										RIBALTINO_DOPO_SQUADRO:
											IF vo = 0 THEN 							
												Mission^.ZPlace			:= 	//WorkArea^[Mission^.PPlace].Z + 
																			Forming^[WorkAreaState^[cwa].F].PackXP[WorkAreaState^[cwa].P].Z + 
																			Forming^[WorkAreaState^[cwa].F].PLZ + 
																			Forming^[WorkAreaState^[cwa].F].PIZ +
																			WorkArea^[Mission^.PPlace].HPL + 
																			HalfPackDim + 
																			ZOffsetPlace + 
																			PickPlaceParameters^.OffsetZPlacePaccoVerticale +
																			DifferenceRealNominalDimensionZ/2;
											(* Quota di deposito Z con pacco orrizontale *)	
											ELSE
												Mission^.ZPlace			:= 	//WorkArea^[Mission^.PPlace].Z + 
																			Forming^[WorkAreaState^[cwa].F].PackXP[WorkAreaState^[cwa].P].Z + 
																			Forming^[WorkAreaState^[cwa].F].PLZ + 
																			WorkArea^[Mission^.PPlace].HPL + 
																			HalfPackDim + 
																			ZOffsetPlace + 
																			PickPlaceParameters^.OffsetZPlacePaccoOrrizzontale;
																			//DifferenceRealNominalDimensionZ/2;
											END_IF
									
										RIBALTINO_DIRETTO:
											IF vo = 0 THEN 							
												Mission^.ZPlace			:= 	//WorkArea^[Mission^.PPlace].Z + 
																			Forming^[WorkAreaState^[cwa].F].PackXP[WorkAreaState^[cwa].P].Z + 
																			Forming^[WorkAreaState^[cwa].F].PLZ + 
																			Forming^[WorkAreaState^[cwa].F].PIZ +
																			WorkArea^[Mission^.PPlace].HPL + 
																			Mission^.XDiM/2 + 
																			ZOffsetPlace + 
																			PickPlaceParameters^.OffsetZPlacePaccoVerticale +
																			DifferenceRealNominalDimensionZ/2;
											(* Quota di deposito Z con pacco orrizontale *)	
											ELSE
												Mission^.ZPlace			:= 	//WorkArea^[Mission^.PPlace].Z + 
																			Forming^[WorkAreaState^[cwa].F].PackXP[WorkAreaState^[cwa].P].Z + 
																			Forming^[WorkAreaState^[cwa].F].PLZ + 
																			WorkArea^[Mission^.PPlace].HPL + 
																			Mission^.ZDim/2 + 
																			ZOffsetPlace + 
																			PickPlaceParameters^.OffsetZPlacePaccoOrrizzontale +
																			DifferenceRealNominalDimensionZ/2;
											END_IF
									END_CASE
									//Mission^.ZPlace			:= WorkArea^[Mission^.PPlace].Z + Forming^[WorkAreaState^[cwa].F].PackXN[WorkAreaState^[cwa].P].Z*2 + WorkArea^[Mission^.PPlace].H;
									Mission^.JPlace			:= 	WorkArea^[Mission^.PPlace].J + 
																WorkAreaOffset^[Mission^.PPlace].J + 
																Forming^[WorkAreaState^[cwa].F].PackXP[WorkAreaState^[cwa].P].J-
																(90*(1-JP)); //x deposito con prelievo TRASVERSALE
									CASE VERSO_PALLETTIZZATORE OF 
										
										PALLETTIZZATORE_DX:
											Mission^.JPlace	:= 	WorkArea^[Mission^.PPlace].J + 
																WorkAreaOffset^[Mission^.PPlace].J + 
																Forming^[WorkAreaState^[cwa].F].PackXP[WorkAreaState^[cwa].P].J-
																(90*(1-JP));
														
										PALLETTIZZATORE_SX:
											Mission^.JPlace	:= 	WorkArea^[Mission^.PPlace].J + 
																WorkAreaOffset^[Mission^.PPlace].J + 
																Forming^[WorkAreaState^[cwa].F].PackXP[WorkAreaState^[cwa].P].J-
																(90*(1-JP));

									END_CASE							
																
																
									IF NOT SimulazioneSenzaPallet THEN //Se non sono in simulazione utilizzo la presa con coppia							
										Mission^.KPlace			:= 	kpick; (*+ 
																PickPlaceParameters^.OffsetKPlacePack;*) // Aggiungere Eventuale Offset x Apertura e Rilascio
									ELSE
										Mission^.KPlace			:= 	kpick + PickPlaceParameters^.OffsetKPickPack;
									END_IF
									Mission^.KPlaceMode 	:= 	KTORQUEMODE;
									(* Quota di Approccio con pacco verticale *)							
									IF (vo = 0 AND DisabilitaApproccioPacciOrrizzontali) OR NOT DisabilitaApproccioPacciOrrizzontali THEN 
										IF  Forming^[WorkAreaState^[cwa].F].PackXP[WorkAreaState^[cwa].P].Trajectory = 0 THEN
											Mission^.XPlaceApproach	:= Mission^.XPlace;
											Mission^.YPlaceApproach	:= Mission^.YPlace;
											Mission^.ZPlaceApproach	:= Mission^.ZPlace;
											Mission^.JPlaceApproach	:= Mission^.JPlace;
										ELSIF  Forming^[WorkAreaState^[cwa].F].PackXP[WorkAreaState^[cwa].P].Trajectory = 1 THEN	
											Mission^.XPlaceApproach	:= 	Mission^.XPlace - 
																		Forming^[WorkAreaState^[cwa].F].AX;
											Mission^.YPlaceApproach	:= 	Mission^.YPlace - 
																		Forming^[WorkAreaState^[cwa].F].AY;
											Mission^.ZPlaceApproach	:= 	Mission^.ZPlace + 
																		Forming^[WorkAreaState^[cwa].F].AZ;
											Mission^.JPlaceApproach	:= 	Mission^.JPlace;
										ELSIF  Forming^[WorkAreaState^[cwa].F].PackXP[WorkAreaState^[cwa].P].Trajectory = 111 THEN	
											Mission^.XPlaceApproach	:= 	Mission^.XPlace - 
																		Forming^[WorkAreaState^[cwa].F].AX;
											Mission^.YPlaceApproach	:= 	Mission^.YPlace - 
																		Forming^[WorkAreaState^[cwa].F].AY;
											Mission^.ZPlaceApproach	:= 	Mission^.ZPlace + 
																		Forming^[WorkAreaState^[cwa].F].AZ;
											Mission^.JPlaceApproach	:= 	Mission^.JPlace;
										ELSIF  Forming^[WorkAreaState^[cwa].F].PackXP[WorkAreaState^[cwa].P].Trajectory = 2 THEN	
											Mission^.XPlaceApproach	:= 	Mission^.XPlace + 
																		Forming^[WorkAreaState^[cwa].F].AX;
											Mission^.YPlaceApproach	:= 	Mission^.YPlace - 
																		Forming^[WorkAreaState^[cwa].F].AY;
											Mission^.ZPlaceApproach	:= 	Mission^.ZPlace + 
																		Forming^[WorkAreaState^[cwa].F].AZ;
											Mission^.JPlaceApproach	:= 	Mission^.JPlace;
										ELSIF  Forming^[WorkAreaState^[cwa].F].PackXP[WorkAreaState^[cwa].P].Trajectory = 101 THEN	
											Mission^.XPlaceApproach	:= 	Mission^.XPlace + 
																		Forming^[WorkAreaState^[cwa].F].AX;
											Mission^.YPlaceApproach	:= 	Mission^.YPlace - 
																		Forming^[WorkAreaState^[cwa].F].AY;
											Mission^.ZPlaceApproach	:= 	Mission^.ZPlace + 
																		Forming^[WorkAreaState^[cwa].F].AZ;
											Mission^.JPlaceApproach	:= 	Mission^.JPlace;
										ELSIF  Forming^[WorkAreaState^[cwa].F].PackXP[WorkAreaState^[cwa].P].Trajectory = 101 THEN	
											Mission^.XPlaceApproach	:= 	Mission^.XPlace + 
																		Forming^[WorkAreaState^[cwa].F].AX;
											Mission^.YPlaceApproach	:= 	Mission^.YPlace - 
																		Forming^[WorkAreaState^[cwa].F].AY;
											Mission^.ZPlaceApproach	:= 	Mission^.ZPlace + 
																		Forming^[WorkAreaState^[cwa].F].AZ;
											Mission^.JPlaceApproach	:= 	Mission^.JPlace;
										ELSIF  Forming^[WorkAreaState^[cwa].F].PackXP[WorkAreaState^[cwa].P].Trajectory = 201 THEN	
											Mission^.XPlaceApproach	:= 	Mission^.XPlace - 
																		Forming^[WorkAreaState^[cwa].F].AX;
											Mission^.YPlaceApproach	:= 	Mission^.YPlace + 
																		Forming^[WorkAreaState^[cwa].F].AY;
											Mission^.ZPlaceApproach	:= 	Mission^.ZPlace + 
																		Forming^[WorkAreaState^[cwa].F].AZ;
											Mission^.JPlaceApproach	:= 	Mission^.JPlace;	
										ELSIF  Forming^[WorkAreaState^[cwa].F].PackXP[WorkAreaState^[cwa].P].Trajectory = 4 THEN	
											Mission^.XPlaceApproach	:= 	Mission^.XPlace + 
																		Forming^[WorkAreaState^[cwa].F].AX;
											Mission^.YPlaceApproach	:= 	Mission^.YPlace + 
																		Forming^[WorkAreaState^[cwa].F].AY;
											Mission^.ZPlaceApproach	:= 	Mission^.ZPlace + 
																		Forming^[WorkAreaState^[cwa].F].AZ;
											Mission^.JPlaceApproach	:= 	Mission^.JPlace;
										ELSIF Forming^[WorkAreaState^[cwa].F].PackXP[WorkAreaState^[cwa].P].Trajectory = 5 THEN	//Esterno-Interno Direzione Y !!!!!!!!!
											Mission^.XPlaceApproach	:= 	Mission^.XPlace;
											IF (Mission^.JPlace = 90 OR Mission^.JPlace = 270) AND Mission^.YPlace >= (WorkArea^[Mission^.PPlace].Y + Pallet^[Workarea^[Mission^.PPlace].Pallet].Y/2) THEN
												Mission^.YPlaceApproach	:= 	Mission^.YPlace + 
																		Forming^[WorkAreaState^[cwa].F].AY;
											ELSE
												Mission^.YPlaceApproach	:= 	Mission^.YPlace - 
																		Forming^[WorkAreaState^[cwa].F].AY;
											END_IF
											Mission^.ZPlaceApproach	:= 	Mission^.ZPlace;
											Mission^.JPlaceApproach	:= 	Mission^.JPlace; 
										ELSIF Forming^[WorkAreaState^[cwa].F].PackXP[WorkAreaState^[cwa].P].Trajectory = 11 THEN	//Esterno-Interno Direzione Y !!!!!!!!!
											Mission^.XPlaceApproach	:= 	Mission^.XPlace;
											IF (Mission^.JPlace = 90 OR Mission^.JPlace = 270) AND Mission^.YPlace >= (WorkArea^[Mission^.PPlace].Y + Pallet^[Workarea^[Mission^.PPlace].Pallet].Y/2) THEN
												Mission^.YPlaceApproach	:= 	Mission^.YPlace + 
																		Forming^[WorkAreaState^[cwa].F].AY;
											ELSE
												Mission^.YPlaceApproach	:= 	Mission^.YPlace - 
																		Forming^[WorkAreaState^[cwa].F].AY;
											END_IF
											Mission^.ZPlaceApproach	:= 	Mission^.ZPlace;
											Mission^.JPlaceApproach	:= 	Mission^.JPlace;
										ELSIF Forming^[WorkAreaState^[cwa].F].PackXP[WorkAreaState^[cwa].P].Trajectory = 21 THEN	//Esterno-Interno Direzione Y !!!!!!!!!
											Mission^.XPlaceApproach	:= 	Mission^.XPlace;
											IF (Mission^.JPlace = 90 OR Mission^.JPlace = 270) AND Mission^.YPlace >= (WorkArea^[Mission^.PPlace].Y + Pallet^[Workarea^[Mission^.PPlace].Pallet].Y/2) THEN
												Mission^.YPlaceApproach	:= 	Mission^.YPlace + 
																		Forming^[WorkAreaState^[cwa].F].AY;
											ELSE
												Mission^.YPlaceApproach	:= 	Mission^.YPlace - 
																		Forming^[WorkAreaState^[cwa].F].AY;
											END_IF
											Mission^.ZPlaceApproach	:= 	Mission^.ZPlace;
											Mission^.JPlaceApproach	:= 	Mission^.JPlace;
										END_IF	
									ELSIF DisabilitaApproccioPacciOrrizzontali and vo = 1 THEN
										Mission^.XPlaceApproach	:= Mission^.XPlace;
										Mission^.YPlaceApproach	:= Mission^.YPlace;
										IF NOT AbilitaDepositoPaccoOrrizzonataleConTasteggio^ THEN
											Mission^.ZPlaceApproach	:= Mission^.ZPlace;
										ELSE
											Mission^.ZPlaceApproach	:= Mission^.ZPlace + QuotaFittizziaPerTasteggioDepPacchi;
										END_IF
										
										Mission^.JPlaceApproach	:= Mission^.JPlace;	
									END_IF
								END_IF
								(* Setto l'uscita che mi determina il deposito del primo pacco in lenta *)
								IF WorkArea^[Mission^.PPlace].Slow = 1 THEN
									DepositoPaccoInLenta := TRUE;
								END_IF
								
								
								WorkAreaManager^.State 	:= WAMANAGER_CICLO_PRELIEVO_PACCO_RUN;
								WAAssegnazionePaccoNONok := FALSE;
							ELSE
								WAAssegnazionePaccoNONok := TRUE;
							END_IF
							
						WAMANAGER_CICLO_PRELIEVO_PACCO_RUN:
							IF Mission^.State = MISSION_STATE_PRELIEVO_PACCO_RUN THEN
								;
							ELSIF Mission^.State = MISSION_STATE_PRELIEVO_PACCO_END THEN
								WorkAreaManager^.State 	:= WAMANAGER_CICLO_PRELIEVO_PACCO_END;
							ELSIF Mission^.State = MISSION_STATE_ERROR THEN
								;
							ELSIF Mission^.State = MISSION_STATE_NOP AND (NOT HandlingRun OR WorkPickPointState^[Mission^.PPick].TS <> WorkPickPointState^[Mission^.PPick].TC) THEN
								WorkAreaManager^.State 	:= WAMANAGER_NOP;
							END_IF	
						
						WAMANAGER_CICLO_PRELIEVO_PACCO_END:	
							(* Copio Info Pacco da Ribaltino a Pinza *)
							Mission^.Pack := TilterPack^;
							RestoreCWA^ := TRUE;
							PreviousPWA^ := pwa;
							//TFPalletizerSetWPPState(WorkPickPointState,Mission^.PPick,WORKPICKPOINT_PRODOTTO_ASSENTE);
							WorkAreaManager^.State 	:= WAMANAGER_CICLO_DEPOSITO_PACCO_RUN;
							ForzaPrelievoPaccoDuranteCicloDiRiposo := FALSE;	
							
						WAMANAGER_CICLO_DEPOSITO_PACCO_RUN:	
							IF Mission^.State = MISSION_STATE_DEPOSITO_PACCO_RUN THEN
								;
							ELSIF Mission^.State = MISSION_STATE_DEPOSITO_PACCO_END THEN
								RestoreCWA^ := TRUE;
								PreviousPWA^ := pwa;
								WorkAreaManager^.State 	:= WAMANAGER_CICLO_DEPOSITO_PACCO_END;	// setto lo stato del WAMANAGER
							END_IF
						
						WAMANAGER_CICLO_DEPOSITO_PACCO_END:
						
							(* Se era settata la velocità lenta di deposito pacco, questa viene resettata *)
							IF WorkArea^[Mission^.PPlace].Slow = 1 THEN
								WorkArea^[Mission^.PPlace].Slow := 0;
								DepositoPaccoInLenta := FALSE;
							END_IF
						
							IF Mission^.TPick = TPICK_PACK THEN
								FOR i:=1 TO MAXHANDLINGSTACK DO
									WorkAreaState^[Mission^.PPlace].Pack[WorkAreaState^[Mission^.PPlace].P,i] := Mission^.Pack[i];
								END_FOR	
							END_IF
						
							(* Punto alla tabella Formatura per verificare se dopo questo pacco devo gestire una Falda *)
							(* La fine formatura la verifico con i dati -1 *)
							IF Forming^[WorkAreaState^[Mission^.PPlace].F].PackXP[WorkAreaState^[Mission^.PPlace].P].Layer > 0 THEN			// se dopo aver depositato un pacco, questo richiede il deposito di una falda (.Layer > 0)
								WorkAreaState^[Mission^.PPlace].L := 0;															// metto a 0 lo stato del layer della piazzola in modo che il manager al ciclo successivo si acorg che bisogna compiere un ciclo falda
								(* Aggiorno Altezza Pallet su Ultimo Pacco *)
								IF Mission^.TPick = TPICK_PACK THEN													// Controllo che la missione  appena eseguita era un prelievo pacco ( dovrebbe sempre essere così!! mantenuto da vecchia gestione..)
									CASE TIPO_RIBALTINO OF
										RIBALTINO_DOPO_SQUADRO:
											IF Forming^[WorkAreaState^[Mission^.PPlace].F].PackXP[WorkAreaState^[Mission^.PPlace].P].Grip = 0 THEN	// Aggiornamento altezza pallet con pacco in verticale (si considera la dimensione Y del pacco) 
												WorkArea^[Mission^.PPlace].H := WorkArea^[Mission^.PPlace].HPL +												// Altezza pallet + layers utilizzati
																	Forming^[WorkAreaState^[Mission^.PPlace].F].PackXP[WorkAreaState^[Mission^.PPlace].P].Z + 	// Quota "Z" del centro del pacco sulla piazzola, cioè altezza assoluta del baricentro
																	Mission^.YDim/2;													//Dimensione Y /2, indica la distanza dal baricentro al bordo superiore del pacco
											ELSIF Forming^[WorkAreaState^[cwa].F].PackXP[WorkAreaState^[cwa].P].Grip = 1 THEN
												WorkArea^[Mission^.PPlace].H := WorkArea^[Mission^.PPlace].HPL + 												// Altezza pallet + layers utilizzati
																	Forming^[WorkAreaState^[Mission^.PPlace].F].PackXP[WorkAreaState^[Mission^.PPlace].P].Z + 	// Quota "Z" del centro del pacco sulla piazzola, cioè altezza assoluta del baricentro
																	Mission^.ZDim/2;													//Dimensione Z /2, indica la distanza dal baricentro al bordo superiore del pacco
											END_IF
											
										RIBALTINO_DIRETTO:
										
											IF Forming^[WorkAreaState^[Mission^.PPlace].F].PackXP[WorkAreaState^[Mission^.PPlace].P].Grip = 0 THEN	// Aggiornamento altezza pallet con pacco in verticale (si considera la dimensione Y del pacco) 
												WorkArea^[Mission^.PPlace].H := WorkArea^[Mission^.PPlace].HPL +												// Altezza pallet + layers utilizzati
																	Forming^[WorkAreaState^[Mission^.PPlace].F].PackXP[WorkAreaState^[Mission^.PPlace].P].Z + 	// Quota "Z" del centro del pacco sulla piazzola, cioè altezza assoluta del baricentro
																	Mission^.XDim/2;													//Dimensione Y /2, indica la distanza dal baricentro al bordo superiore del pacco
											ELSIF Forming^[WorkAreaState^[cwa].F].PackXP[WorkAreaState^[cwa].P].Grip = 1 THEN
												WorkArea^[Mission^.PPlace].H := WorkArea^[Mission^.PPlace].HPL + 												// Altezza pallet + layers utilizzati
																	Forming^[WorkAreaState^[Mission^.PPlace].F].PackXP[WorkAreaState^[Mission^.PPlace].P].Z + 	// Quota "Z" del centro del pacco sulla piazzola, cioè altezza assoluta del baricentro
																	Mission^.ZDim/2;													//Dimensione Z /2, indica la distanza dal baricentro al bordo superiore del pacco
											END_IF
									END_CASE
								END_IF
								RestoreCWA^ := TRUE;
								PreviousPWA^ := pwa;
								WorkAreaManager^.State 	:= WAMANAGER_NOP;	// setto lo stato del WAMANAGER
								EXIT;
							ELSE																								// se dopo aver depositato un pacco, NON DEVO depositare NESSUNA falda
								(* Aggiorno Altezza Pallet su Ultimo Pacco *)
								IF Mission^.TPick = TPICK_PACK THEN													// Controllo che la missione  appena eseguita era un prelievo pacco ( dovrebbe sempre essere così!! mantenuto da vecchia gestione..)
									CASE TIPO_RIBALTINO OF
										RIBALTINO_DOPO_SQUADRO:
											IF Forming^[WorkAreaState^[Mission^.PPlace].F].PackXP[WorkAreaState^[Mission^.PPlace].P].Grip = 0 THEN	// Aggiornamento altezza pallet con pacco in verticale (si considera la dimensione Y del pacco) 
												WorkArea^[Mission^.PPlace].H := WorkArea^[Mission^.PPlace].HPL +												// Altezza pallet + layers utilizzati
																	Forming^[WorkAreaState^[Mission^.PPlace].F].PackXP[WorkAreaState^[Mission^.PPlace].P].Z + 	// Quota "Z" del centro del pacco sulla piazzola, cioè altezza assoluta del baricentro
																	Mission^.YDim/2;													//Dimensione Y /2, indica la distanza dal baricentro al bordo superiore del pacco
											ELSIF Forming^[WorkAreaState^[cwa].F].PackXP[WorkAreaState^[cwa].P].Grip = 1 THEN
												WorkArea^[Mission^.PPlace].H := WorkArea^[Mission^.PPlace].HPL + 												// Altezza pallet + layers utilizzati
																	Forming^[WorkAreaState^[Mission^.PPlace].F].PackXP[WorkAreaState^[Mission^.PPlace].P].Z + 	// Quota "Z" del centro del pacco sulla piazzola, cioè altezza assoluta del baricentro
																	Mission^.ZDim/2;													//Dimensione Z /2, indica la distanza dal baricentro al bordo superiore del pacco
											END_IF
											
										RIBALTINO_DIRETTO:
										
											IF Forming^[WorkAreaState^[Mission^.PPlace].F].PackXP[WorkAreaState^[Mission^.PPlace].P].Grip = 0 THEN	// Aggiornamento altezza pallet con pacco in verticale (si considera la dimensione Y del pacco) 
												WorkArea^[Mission^.PPlace].H := WorkArea^[Mission^.PPlace].HPL +												// Altezza pallet + layers utilizzati
																	Forming^[WorkAreaState^[Mission^.PPlace].F].PackXP[WorkAreaState^[Mission^.PPlace].P].Z + 	// Quota "Z" del centro del pacco sulla piazzola, cioè altezza assoluta del baricentro
																	Mission^.XDim/2;													//Dimensione Y /2, indica la distanza dal baricentro al bordo superiore del pacco
											ELSIF Forming^[WorkAreaState^[cwa].F].PackXP[WorkAreaState^[cwa].P].Grip = 1 THEN
												WorkArea^[Mission^.PPlace].H := WorkArea^[Mission^.PPlace].HPL + 												// Altezza pallet + layers utilizzati
																	Forming^[WorkAreaState^[Mission^.PPlace].F].PackXP[WorkAreaState^[Mission^.PPlace].P].Z + 	// Quota "Z" del centro del pacco sulla piazzola, cioè altezza assoluta del baricentro
																	Mission^.ZDim/2;													//Dimensione Z /2, indica la distanza dal baricentro al bordo superiore del pacco
											END_IF
									END_CASE
								END_IF
								(* Incremento WorkArea^[cwa].P (P=P+1) *)
								WorkAreaState^[Mission^.PPlace].P := WorkAreaState^[Mission^.PPlace].P + 1;
								(* Controllo Fine Pallettizzazione o Deposito Falda Dopo Strato Pacchi*)
								(* COME FACCIO A SAPERE SE è L'ULTIMO PACCO ? -> Si controlla la Grip=-1 *)
								(* Per sicurezza le controllo su entrambi le direzioni POSITIVA/NEGATIVA *)
								IF Forming^[WorkAreaState^[Mission^.PPlace].F].PackXP[WorkAreaState^[Mission^.PPlace].P].Grip = -1 OR
									Forming^[WorkAreaState^[Mission^.PPlace].F].PackXN[WorkAreaState^[Mission^.PPlace].P].Grip = -1 THEN
									IF NOT BypassTEST AND TRUE THEN //se true inizializza la piazzola a 1 pacco una volta completata la pallettizzazione
										WorkAreaState^[Mission^.PPlace].State := WORKAREA_STATE_OCCUPIED_WORKED;
										WorkAreaManager^.State 	:= WAMANAGER_NOP;	// setto lo stato del WAMANAGER
										RestoreCWA^ := TRUE;
										PreviousPWA^ := pwa;
										EXIT;
									ELSE
										WorkAreaState^[Mission^.PPlace].P := 1;
										WorkAreaManager^.State 	:= WAMANAGER_NOP;	// setto lo stato del WAMANAGER
										RestoreCWA^ := TRUE;
										PreviousPWA^ := pwa;
										EXIT;
									END_IF			
								END_IF
								WorkAreaManager^.State 	:= WAMANAGER_NOP;	// setto lo stato del WAMANAGER
								EXIT;
							END_IF								
					END_CASE	//riferito al case WorkAreaManager^.State
				ELSE			// riferito all' IF prima del  case WorkAreaManager^.State
					RestoreCWA^ := TRUE;
					PreviousPWA^ := pwa;
					WorkAreaState^[cwa].State := WORKAREA_STATE_OCCUPIED_DISABLED;
					EXIT;
				END_IF			// riferito all' IF prima del  case WorkAreaManager^.State

(**********************************************************************************************************************************************************************************)
(**********************************************************************************************************************************************************************************)
			(* ******************************************************************************************************** *)
						(* GESTIONE (Nastratura) o (Veicolo per prelievo/deposito PALLET FINITI/CATASTE/FALDE) *)
			(* ******************************************************************************************************** *)
(**********************************************************************************************************************************************************************************)
(**********************************************************************************************************************************************************************************)
			(* Occupied + Worked *)
			WORKAREA_STATE_OCCUPIED_WORKED:
				IF WorkArea^[cwa].Enable = 1 THEN
					IF NOT WorkArea^[cwa].RefuseLGV THEN		
						IF Forming^[WorkAreaState^[cwa].F].Tape = 0 THEN
							WorkAreaState^[cwa].State := WORKAREA_STATE_OCCUPIED_ENDED;
						ELSIF Forming^[WorkAreaState^[cwa].F].Tape = 1 THEN
							WorkAreaState^[cwa].State := WORKAREA_STATE_OCCUPIED_TAPING;
						END_IF
					ELSIF WorkArea^[cwa].RefuseLGV AND WorkArea^[cwa].LGV_Req = 1 THEN
						WorkArea^[cwa].LGV_Req := 0;
					END_IF	
				ELSE
					WorkAreaState^[cwa].State := WORKAREA_STATE_OCCUPIED_WORKED_DISABLED;
				END_IF
	
			(* Occupied + Worked + Disabled *)
			WORKAREA_STATE_OCCUPIED_WORKED_DISABLED:
				WorkArea^[cwa].LGV_Req := 0;
				IF WorkArea^[cwa].Enable = 1 THEN
					WorkAreaState^[cwa].State := WORKAREA_STATE_OCCUPIED_WORKED;
				ELSE
					;
				END_IF
	
			(* Occupied + Taping *)
			WORKAREA_STATE_OCCUPIED_TAPING:
				WorkArea^[cwa].LGV_Req := 0;
				IF WorkArea^[cwa].Enable = 1 THEN
					IF WorkArea^[cwa].LGV_Req = 0 AND  WorkArea^[cwa].LGV_ReqAbort THEN
						WorkAreaState^[cwa].State := WORKAREA_STATE_OCCUPIED_WORKING;
						WorkArea^[cwa].LGV_ReqAbort := FALSE;
					ELSE
						IF WorkArea^[cwa].Taped = 1 OR Forming^[WorkAreaState^[cwa].F].Tape = 0 THEN
							WorkAreaState^[cwa].State := WORKAREA_STATE_OCCUPIED_TAPED;
						END_IF
					END_IF	
				ELSE
					WorkAreaState^[cwa].State := WORKAREA_STATE_OCCUPIED_TAPING_DISABLED;
				END_IF
	
			(* Occupied + Taping + Disabled *)
			WORKAREA_STATE_OCCUPIED_TAPING_DISABLED:
				IF WorkArea^[cwa].Enable = 1 THEN
					WorkAreaState^[cwa].State := WORKAREA_STATE_OCCUPIED_TAPING;
				ELSE
					;
				END_IF
	
			(* Occupied + Taped *)
			WORKAREA_STATE_OCCUPIED_TAPED:
				IF WorkArea^[cwa].Enable = 1 THEN
					WorkAreaState^[cwa].State := WORKAREA_STATE_OCCUPIED_ENDED;
				ELSE
					WorkAreaState^[cwa].State := WORKAREA_STATE_OCCUPIED_TAPED_DISABLED;
				END_IF
	
			(* Occupied + Taped + Disabled *)
			WORKAREA_STATE_OCCUPIED_TAPED_DISABLED:
				WorkArea^[cwa].LGV_Req := 0;
				IF WorkArea^[cwa].Enable = 1 THEN
					WorkAreaState^[cwa].State := WORKAREA_STATE_OCCUPIED_TAPED;
				ELSE
					;
				END_IF
	
			(* Occupied + Ended *)
			WORKAREA_STATE_OCCUPIED_ENDED:
				IF WorkArea^[cwa].Enable = 1 THEN
					IF WorkArea^[cwa].Typology = TYPOLOGY_PALLET OR WorkArea^[cwa].Typology = TYPOLOGY_STACK AND NOT PX_WorkArea[cwa] THEN
						WorkAreaState^[cwa].State := WORKAREA_STATE_OCCUPIED_LGVREQ;
					END_IF	
				ELSE
					WorkAreaState^[cwa].State := WORKAREA_STATE_OCCUPIED_ENDED_DISABLED;
				END_IF
	
			(* Occupied + Ended + Disabled *)
			WORKAREA_STATE_OCCUPIED_ENDED_DISABLED:
				IF WorkArea^[cwa].Enable = 1 THEN
					WorkAreaState^[cwa].State := WORKAREA_STATE_OCCUPIED_ENDED;
				ELSE
					;
				END_IF
	
		 (* (* Occupied + LgvReq *)
			WORKAREA_STATE_OCCUPIED_LGVREQ:
				IF WorkArea^[cwa].Enable = 1 THEN
					; // Gestito dalla FB TFLGV
					IF WorkArea^[cwa].LGV_ReqAbort THEN
						WorkArea^[cwa].LGV_Req := 0;
						WorkArea^[cwa].LGV_ReqAbort := FALSE;
					ELSE
						WorkArea^[cwa].LGV_Req := 1; //aggiunto per comunicazione con LGV
						IF Forming^[WorkAreaState^[cwa].F].Tape = 1 AND WorkArea^[cwa].Taped < 1 THEN
							WorkArea^[cwa].LGV_Req := 0;
							WorkAreaState^[cwa].State := WORKAREA_STATE_OCCUPIED_WORKED;
						END_IF
					END_IF
				ELSE
					WorkAreaState^[cwa].State := WORKAREA_STATE_OCCUPIED_LGVREQ_DISABLED;				
				END_IF*)
				
			(* Occupied + LgvReq *)
			WORKAREA_STATE_OCCUPIED_LGVREQ:
				IF WorkArea^[cwa].Enable = 1 THEN
					IF Forming^[WorkAreaState^[cwa].F].Tape = 1 AND WorkArea^[cwa].Taped < 1 and WorkArea^[cwa].Typology = TYPOLOGY_PALLET THEN
						WorkArea^[cwa].LGV_Req := 0;
						WorkArea^[cwa].LGV_ReqAbort := FALSE;
						WorkAreaState^[cwa].State := WORKAREA_STATE_OCCUPIED_WORKED;
						EXIT;
					END_IF
					IF WorkArea^[cwa].LGV_ReqAbort THEN
						WorkArea^[cwa].LGV_Req := 0;
						WorkAreaState^[cwa].State := WORKAREA_STATE_OCCUPIED_LGVREQ_ABORT;
					ELSIF (NOT WorkArea^[cwa].LGV_ReqAbort AND WorkArea^[cwa].LGV_Req = 0) AND WorkArea^[cwa].Typology = TYPOLOGY_PALLET THEN
						IF Forming^[WorkAreaState^[cwa].F].PackXP[WorkAreaState^[cwa].P].Grip = -1 OR
							Forming^[WorkAreaState^[cwa].F].PackXN[WorkAreaState^[cwa].P].Grip = -1 THEN
							WorkArea^[cwa].LGV_Req := 1; 
						ELSE
							WorkAreaState^[cwa].State := WORKAREA_STATE_OCCUPIED_WORKING;
							EXIT;
						END_IF
					ELSE
						WorkArea^[cwa].LGV_Req := 1; 
					END_IF	
				ELSE
					WorkAreaState^[cwa].State := WORKAREA_STATE_OCCUPIED_LGVREQ_DISABLED;				
				END_IF
	
			(* Occupied + LgvReq + Disabled *)
			WORKAREA_STATE_OCCUPIED_LGVREQ_DISABLED:
				WorkArea^[cwa].LGV_Req := 0;
				IF WorkArea^[cwa].Enable = 1 THEN
					WorkAreaState^[cwa].State := WORKAREA_STATE_OCCUPIED_LGVREQ;
				ELSE
					;
				END_IF
				
			(* Occupied + LgvReqAbort *)
			WORKAREA_STATE_OCCUPIED_LGVREQ_ABORT:
				IF WorkArea^[cwa].Enable = 1 THEN
					IF (Forming^[WorkAreaState^[cwa].F].PackXP[WorkAreaState^[cwa].P].Grip <> -1 OR
						Forming^[WorkAreaState^[cwa].F].PackXN[WorkAreaState^[cwa].P].Grip <> -1) AND WorkArea^[cwa].LGV_ReqAbort THEN
							WorkAreaState^[cwa].State := WORKAREA_STATE_OCCUPIED_WORKING;
							WorkArea^[cwa].LGV_ReqAbort := FALSE;
							EXIT;
					ELSIF WorkArea^[cwa].LGV_ReqAbort THEN
						WorkArea^[cwa].LGV_Req := 0;
						//WorkArea^[cwa].LGV_ReqAbort := FALSE;
						EXIT;
					ELSIF WorkArea^[cwa].LGV_Req = 1 OR (Forming^[WorkAreaState^[cwa].F].PackXP[WorkAreaState^[cwa].P].Grip = -1 OR
						Forming^[WorkAreaState^[cwa].F].PackXN[WorkAreaState^[cwa].P].Grip = -1) THEN
							WorkAreaState^[cwa].State := WORKAREA_STATE_OCCUPIED_LGVREQ; 
							EXIT;
					END_IF
				ELSE
					;
				END_IF
	
			(* Occupied + LgvIn  - NOT USED !!!!!!!!!!!*)
			WORKAREA_STATE_OCCUPIED_LGVIN:
				IF WorkArea^[cwa].Enable = 1 THEN
					;
				ELSE
					;
				END_IF
	
			(* Occupied + LgvIn + Disabled  - NOT USED !!!!!!!!!!!*)
			WORKAREA_STATE_OCCUPIED_LGVIN_DISABLED:
				IF WorkArea^[cwa].Enable = 1 THEN
					;
				ELSE
					;
				END_IF
	
			(* Occupied + LgvEnd  - NOT USED !!!!!!!!!!!*)
			WORKAREA_STATE_OCCUPIED_LGVEND:
				IF WorkArea^[cwa].Enable = 1 THEN
					;
				ELSE
					;
				END_IF
	
			(* Occupied + LgvIn + Disabled - NOT USED !!!!!!!!!!! *)
			WORKAREA_STATE_OCCUPIED_LGVEND_DISABLED:
				IF WorkArea^[cwa].Enable = 1 THEN
					;
				ELSE
					;
				END_IF
	
			(* Error *)
			WORKAREA_STATE_ERROR:
				;
	
		ELSE		//riferito al WorkAreaState^[cwa].State								
			(* Stato Errato. viene Forzato lo stato di errore. Non dovrebbe MAI accadere *)
			WorkAreaState^[cwa].State := WORKAREA_STATE_ERROR;
				
		END_CASE;  //riferito al WorkAreaState^[cwa].State
	
	END_FOR			// riferito a FOR pwa:=1 TO MAXAREA DO


END_IF 				// riferito a IF WaitPositionRequest > 0 AND

//TFPalletizerWorkAreaManagerTF := TRUE;

END_FUNCTION_BLOCK

(* stored: Version 1.1.0.1, ProductVersion 3.1.4024.11
   POU TFPalletizerWorkAreaManagerTF: Id {5aec937a-63b7-4604-9c04-c96d7b224bb2}, SpecialFunc None *)
